Yaskawa INFORM job: ARGAZ.JBI

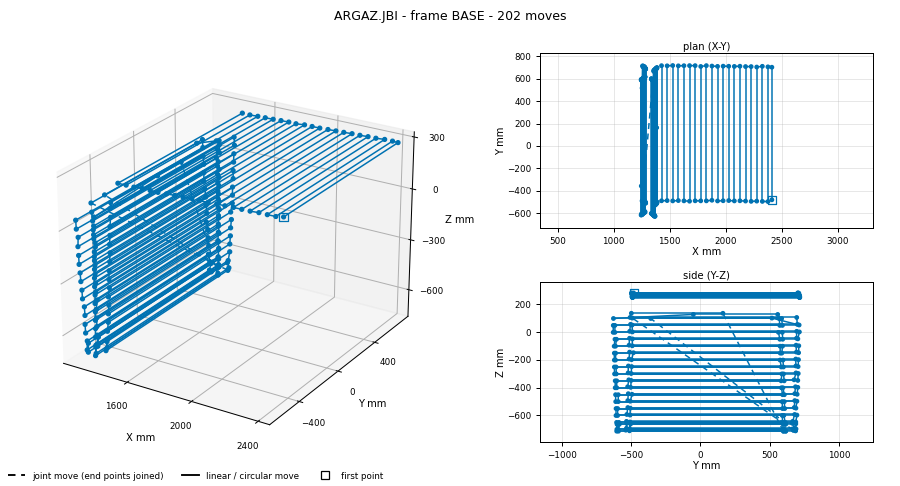
[picture p0: tool path of ARGAZ.JBI in frame BASE, 202 of 208 moves have a stored position in this frame; points joined in program order, loops and branches not executed]
/JOB
//NAME ARGAZ
//POS
///NPOS 202,0,202,0,0,0
///TOOL 0
///POSTYPE BASE
///RECTAN
///RCONF 1,0,0,0,0,0,0,0,0,0,0,0,0,0,0,0,0,0,0,0,0,0,0,0
C00000=2413.206274,-480.697971,282.313473,175.000000,5.000000,5.000000
C00001=2413.206274,703.166336,282.313473,175.000000,5.000000,5.000000
C00002=2378.104531,706.654151,282.437477,175.000000,5.000000,5.000000
C00003=2378.104531,-496.268820,282.437477,175.000000,5.000000,5.000000
C00004=2328.104531,-494.692713,280.280820,175.000000,5.000000,5.000000
C00005=2328.104531,711.367526,280.280820,175.000000,5.000000,5.000000
C00006=2278.104531,704.842987,278.975224,175.000000,5.000000,5.000000
C00007=2278.104531,-492.369314,278.975224,175.000000,5.000000,5.000000
C00008=2228.104531,-494.327219,276.432500,175.000000,5.000000,5.000000
C00009=2228.104531,708.877685,276.432500,175.000000,5.000000,5.000000
C00010=2178.104531,709.094399,273.988824,175.000000,5.000000,5.000000
C00011=2178.104531,-491.808166,273.988824,175.000000,5.000000,5.000000
C00012=2128.104531,-489.305417,272.087718,175.000000,5.000000,5.000000
C00013=2128.104531,712.128405,272.087718,175.000000,5.000000,5.000000
C00014=2078.104531,710.272403,270.104441,175.000000,5.000000,5.000000
C00015=2078.104531,-490.482062,270.104441,175.000000,5.000000,5.000000
C00016=2028.104531,-487.207564,267.676628,175.000000,5.000000,5.000000
C00017=2028.104531,711.894706,267.676628,175.000000,5.000000,5.000000
C00018=1978.104531,712.621618,265.646129,175.000000,5.000000,5.000000
C00019=1978.104531,-488.994271,265.646129,175.000000,5.000000,5.000000
C00020=1928.104531,-490.817664,264.262632,175.000000,5.000000,5.000000
C00021=1928.104531,710.764257,264.262632,175.000000,5.000000,5.000000
C00022=1878.104531,713.606685,262.597692,175.000000,5.000000,5.000000
C00023=1878.104531,-484.609026,262.597692,175.000000,5.000000,5.000000
C00024=1828.104531,-490.014665,260.699234,175.000000,5.000000,5.000000
C00025=1828.104531,717.443690,260.699234,175.000000,5.000000,5.000000
C00026=1778.104531,710.010172,259.433237,175.000000,5.000000,5.000000
C00027=1778.104531,-489.903250,259.433237,175.000000,5.000000,5.000000
C00028=1728.104531,-489.503789,257.000034,175.000000,5.000000,5.000000
C00029=1728.104531,717.230372,257.000034,175.000000,5.000000,5.000000
C00030=1678.104531,717.470864,255.326624,175.000000,5.000000,5.000000
C00031=1678.104531,-493.010626,255.326624,175.000000,5.000000,5.000000
C00032=1628.104531,-489.934501,253.475395,175.000000,5.000000,5.000000
C00033=1628.104531,716.829551,253.475395,175.000000,5.000000,5.000000
C00034=1578.104531,715.609427,252.672152,175.000000,5.000000,5.000000
C00035=1578.104531,-487.412050,252.672152,175.000000,5.000000,5.000000
C00036=1528.104531,-490.348908,250.461753,175.000000,5.000000,5.000000
C00037=1528.104531,718.341799,250.461753,175.000000,5.000000,5.000000
C00038=1478.104531,715.724918,249.387703,175.000000,5.000000,5.000000
C00039=1478.104531,-487.359740,249.387703,175.000000,5.000000,5.000000
C00040=1428.054088,-489.367917,249.591600,175.000000,5.000000,5.000000
C00041=1428.054088,717.087707,249.591600,175.000000,5.000000,5.000000
C00042=1375.381280,558.865130,127.297261,175.000000,-89.999999,5.000000
C00043=1375.381280,-49.872904,127.297261,175.000000,-89.999999,5.000000
C00044=1370.317972,-626.433977,98.135956,175.000000,-89.999999,5.000000
C00045=1370.317972,569.304121,98.135956,175.000000,-89.999999,5.000000
C00046=1368.165956,573.982169,48.135956,175.000000,-89.999999,5.000000
C00047=1368.165956,-627.765516,48.135956,175.000000,-89.999999,5.000000
C00048=1366.300613,-628.336175,-1.864044,175.000000,-89.999999,5.000000
C00049=1366.300613,564.146447,-1.864044,175.000000,-89.999999,5.000000
C00050=1364.709070,574.518860,-51.864044,175.000000,-89.999999,5.000000
C00051=1364.709070,-615.470524,-51.864044,175.000000,-89.999999,5.000000
C00052=1362.699081,-621.338804,-101.864044,175.000000,-89.999999,5.000000
C00053=1362.699081,576.164261,-101.864044,175.000000,-89.999999,5.000000
C00054=1361.029734,577.134382,-151.864044,175.000000,-89.999999,5.000000
C00055=1361.029734,-620.046668,-151.864044,175.000000,-89.999999,5.000000
C00056=1359.409458,-620.048027,-201.864044,175.000000,-89.999999,5.000000
C00057=1359.409458,575.847681,-201.864044,175.000000,-89.999999,5.000000
C00058=1357.613517,584.372245,-251.864044,175.000000,-89.999999,5.000000
C00059=1357.613517,-619.966504,-251.864044,175.000000,-89.999999,5.000000
C00060=1355.809114,-618.285777,-301.864044,175.000000,-89.999999,5.000000
C00061=1355.809114,588.836976,-301.864044,175.000000,-89.999999,5.000000
C00062=1353.972481,583.403483,-351.864044,175.000000,-89.999999,5.000000
C00063=1353.972481,-613.874036,-351.864044,175.000000,-89.999999,5.000000
C00064=1352.018958,-613.863166,-401.864044,175.000000,-89.999999,5.000000
C00065=1352.018958,585.494542,-401.864044,175.000000,-89.999999,5.000000
C00066=1350.088816,594.463405,-451.864044,175.000000,-89.999999,5.000000
C00067=1350.088816,-611.032968,-451.864044,175.000000,-89.999999,5.000000
C00068=1348.161110,-610.087304,-501.864044,175.000000,-89.999999,5.000000
C00069=1348.161110,590.588356,-501.864044,175.000000,-89.999999,5.000000
C00070=1346.094321,593.798995,-551.864044,175.000000,-89.999999,5.000000
C00071=1346.094321,-607.729937,-551.864044,175.000000,-89.999999,5.000000
C00072=1344.309797,-608.197334,-601.864044,175.000000,-89.999999,5.000000
C00073=1344.309797,591.908346,-601.864044,175.000000,-89.999999,5.000000
C00074=1342.380235,593.679428,-651.864044,175.000000,-89.999999,5.000000
C00075=1342.380235,-603.654478,-651.864044,175.000000,-89.999999,5.000000
C00076=1340.669129,-601.653773,-701.864044,175.000000,-89.999999,5.000000
C00077=1340.669129,595.156349,-701.864044,175.000000,-89.999999,5.000000
C00078=1338.968924,598.160463,-665.261503,180.000000,-60.000000,0.000000
C00079=1338.968924,-600.617076,-665.261503,180.000000,-60.000000,0.000000
C00080=1337.538666,-602.949985,-715.261503,180.000000,-60.000000,0.000000
C00081=1337.538666,600.315381,-715.261503,180.000000,-60.000000,0.000000
C00082=1337.538666,600.315381,-715.261503,180.000000,-60.000000,0.000000
C00083=1384.573264,163.476492,135.649179,175.000000,-89.999999,5.000000
C00084=1384.573264,-497.212784,135.649179,175.000000,-89.999999,5.000000
C00085=1387.134154,-506.685611,105.452428,175.000000,-89.999999,5.000000
C00086=1387.134154,696.005872,105.452428,175.000000,-89.999999,5.000000
C00087=1386.644943,700.400566,55.452428,175.000000,-89.999999,5.000000
C00088=1386.644943,-503.175845,55.452428,175.000000,-89.999999,5.000000
C00089=1385.416341,-509.347205,5.452428,175.000000,-89.999999,5.000000
C00090=1385.416341,695.993619,5.452428,175.000000,-89.999999,5.000000
C00091=1384.530286,694.673032,-44.547572,175.000000,-89.999999,5.000000
C00092=1384.530286,-510.215797,-44.547572,175.000000,-89.999999,5.000000
C00093=1383.211942,-513.702418,-94.547572,175.000000,-89.999999,5.000000
C00094=1383.211942,691.424661,-94.547572,175.000000,-89.999999,5.000000
C00095=1382.029329,693.773127,-144.547572,175.000000,-89.999999,5.000000
C00096=1382.029329,-510.105522,-144.547572,175.000000,-89.999999,5.000000
C00097=1380.742282,-513.419241,-194.547572,175.000000,-89.999999,5.000000
C00098=1380.742282,689.151074,-194.547572,175.000000,-89.999999,5.000000
C00099=1379.317619,689.923005,-244.547572,175.000000,-89.999999,5.000000
C00100=1379.317619,-518.588589,-244.547572,175.000000,-89.999999,5.000000
C00101=1377.622991,-520.482337,-294.547572,175.000000,-89.999999,5.000000
C00102=1377.622991,690.843331,-294.547572,175.000000,-89.999999,5.000000
C00103=1375.725701,676.986701,-344.547572,175.000000,-89.999999,5.000000
C00104=1375.725701,-515.830333,-344.547572,175.000000,-89.999999,5.000000
C00105=1373.930863,-523.962151,-394.547572,175.000000,-89.999999,5.000000
C00106=1373.930863,687.201507,-394.547572,175.000000,-89.999999,5.000000
C00107=1371.931878,682.022629,-444.547572,175.000000,-89.999999,5.000000
C00108=1371.931878,-519.291087,-444.547572,175.000000,-89.999999,5.000000
C00109=1370.288163,-523.069053,-494.547572,175.000000,-89.999999,5.000000
C00110=1370.288163,681.905546,-494.547572,175.000000,-89.999999,5.000000
C00111=1368.373992,678.466575,-544.547572,175.000000,-89.999999,5.000000
C00112=1368.373992,-522.809020,-544.547572,175.000000,-89.999999,5.000000
C00113=1366.288380,-529.990561,-594.547572,175.000000,-89.999999,5.000000
C00114=1366.288380,681.080520,-594.547572,175.000000,-89.999999,5.000000
C00115=1364.367259,667.085024,-644.547572,175.000000,-89.999999,5.000000
C00116=1364.367259,-532.326774,-644.547572,175.000000,-89.999999,5.000000
C00117=1362.423936,-532.694360,-694.547572,175.000000,-89.999999,5.000000
C00118=1362.423936,677.683753,-694.547572,175.000000,-89.999999,5.000000
C00119=1360.448293,664.032699,-657.945032,180.000000,-60.000000,0.000000
C00120=1360.448293,-528.686312,-657.945032,180.000000,-60.000000,0.000000
C00121=1358.736655,-537.636349,-707.945032,180.000000,-60.000000,0.000000
C00122=1358.736655,671.519200,-707.945032,180.000000,-60.000000,0.000000
C00123=1358.736655,671.519200,-707.945032,180.000000,-60.000000,0.000000
C00124=1254.346646,-489.805456,101.042867,175.000000,-89.999999,5.000000
C00125=1254.346646,517.104174,101.042867,175.000000,-89.999999,5.000000
C00126=1258.463174,713.476215,51.042867,175.000000,-89.999999,5.000000
C00127=1258.463174,-491.860509,51.042867,175.000000,-89.999999,5.000000
C00128=1261.233179,-489.734803,1.042867,175.000000,-89.999999,5.000000
C00129=1261.233179,715.246618,1.042867,175.000000,-89.999999,5.000000
C00130=1263.530822,704.150010,-48.957133,175.000000,-89.999999,5.000000
C00131=1263.530822,-489.611160,-48.957133,175.000000,-89.999999,5.000000
C00132=1265.803484,-490.551389,-98.957133,175.000000,-89.999999,5.000000
C00133=1265.803484,711.067217,-98.957133,175.000000,-89.999999,5.000000
C00134=1268.209382,709.711222,-148.957133,175.000000,-89.999999,5.000000
C00135=1268.209382,-482.270035,-148.957133,175.000000,-89.999999,5.000000
C00136=1269.839575,-495.608518,-198.957133,175.000000,-89.999999,5.000000
C00137=1269.839575,708.751971,-198.957133,175.000000,-89.999999,5.000000
C00138=1271.633535,706.020958,-248.957133,175.000000,-89.999999,5.000000
C00139=1271.633535,-495.046011,-248.957133,175.000000,-89.999999,5.000000
C00140=1273.209045,-498.528392,-298.957133,175.000000,-89.999999,5.000000
C00141=1273.209045,707.091624,-298.957133,175.000000,-89.999999,5.000000
C00142=1274.778950,703.821202,-348.957133,175.000000,-89.999999,5.000000
C00143=1274.778950,-498.652035,-348.957133,175.000000,-89.999999,5.000000
C00144=1276.502901,-501.906152,-398.957133,175.000000,-89.999999,5.000000
C00145=1276.502901,703.989682,-398.957133,175.000000,-89.999999,5.000000
C00146=1277.998844,699.262721,-448.957133,175.000000,-89.999999,5.000000
C00147=1277.998844,-492.101681,-448.957133,175.000000,-89.999999,5.000000
C00148=1279.424846,-505.182009,-498.957133,175.000000,-89.999999,5.000000
C00149=1279.424846,697.394490,-498.957133,175.000000,-89.999999,5.000000
C00150=1280.126954,690.352282,-548.957133,175.000000,-89.999999,5.000000
C00151=1280.126954,-504.584175,-548.957133,175.000000,-89.999999,5.000000
C00152=1281.384025,-506.767627,-598.957133,175.000000,-89.999999,5.000000
C00153=1281.384025,697.495035,-598.957133,175.000000,-89.999999,5.000000
C00154=1282.818366,689.325095,-648.957133,175.000000,-89.999999,5.000000
C00155=1282.818366,-506.682028,-648.957133,175.000000,-89.999999,5.000000
C00156=1284.126716,-509.875003,-698.957133,175.000000,-89.999999,5.000000
C00157=1284.126716,691.027562,-698.957133,175.000000,-89.999999,5.000000
C00158=1285.461074,689.375368,-662.354593,180.000000,-60.000000,0.000000
C00159=1285.461074,-501.749900,-662.354593,180.000000,-60.000000,0.000000
C00160=1286.533597,-510.586968,-712.354593,180.000000,-60.000000,0.000000
C00161=1286.533597,687.223167,-712.354593,180.000000,-60.000000,0.000000
C00162=1286.533597,687.223167,-712.354593,180.000000,-60.000000,0.000000
C00163=1247.184948,-357.258152,98.133703,175.000000,-89.999999,5.000000
C00164=1247.184948,587.097994,98.133703,175.000000,-89.999999,5.000000
C00165=1245.843306,592.746565,48.133703,175.000000,-89.999999,5.000000
C00166=1245.843306,-616.020977,48.133703,175.000000,-89.999999,5.000000
C00167=1247.718409,-615.852160,-1.866297,175.000000,-89.999999,5.000000
C00168=1247.718409,592.113501,-1.866297,175.000000,-89.999999,5.000000
C00169=1249.627062,594.663458,-51.866297,175.000000,-89.999999,5.000000
C00170=1249.627062,-604.746979,-51.866297,175.000000,-89.999999,5.000000
C00171=1251.401209,-611.430237,-101.866297,175.000000,-89.999999,5.000000
C00172=1251.401209,593.745855,-101.866297,175.000000,-89.999999,5.000000
C00173=1253.367892,588.365485,-151.866297,175.000000,-89.999999,5.000000
C00174=1253.367892,-610.535777,-151.866297,175.000000,-89.999999,5.000000
C00175=1255.139335,-611.488778,-201.866297,175.000000,-89.999999,5.000000
C00176=1255.139335,597.021454,-201.866297,175.000000,-89.999999,5.000000
C00177=1256.999427,599.889986,-251.866297,175.000000,-89.999999,5.000000
C00178=1256.999427,-607.499790,-251.866297,175.000000,-89.999999,5.000000
C00179=1259.062129,-606.254082,-301.866297,175.000000,-89.999999,5.000000
C00180=1259.062129,600.841625,-301.866297,175.000000,-89.999999,5.000000
C00181=1261.582176,605.514051,-351.866297,175.000000,-89.999999,5.000000
C00182=1261.582176,-602.829406,-351.866297,175.000000,-89.999999,5.000000
C00183=1263.639717,-602.839616,-401.866297,175.000000,-89.999999,5.000000
C00184=1263.639717,596.578989,-401.866297,175.000000,-89.999999,5.000000
C00185=1265.975009,606.745464,-451.866297,175.000000,-89.999999,5.000000
C00186=1265.975009,-591.829736,-451.866297,175.000000,-89.999999,5.000000
C00187=1268.177807,-591.867856,-501.866297,175.000000,-89.999999,5.000000
C00188=1268.177807,606.511299,-501.866297,175.000000,-89.999999,5.000000
C00189=1270.115574,609.444498,-551.866297,175.000000,-89.999999,5.000000
C00190=1270.115574,-596.282972,-551.866297,175.000000,-89.999999,5.000000
C00191=1272.145767,-596.372826,-601.866297,175.000000,-89.999999,5.000000
C00192=1272.145767,602.765325,-601.866297,175.000000,-89.999999,5.000000
C00193=1274.380461,613.267393,-651.866297,175.000000,-89.999999,5.000000
C00194=1274.380461,-586.885024,-651.866297,175.000000,-89.999999,5.000000
C00195=1276.674662,-593.241538,-701.866297,175.000000,-89.999999,5.000000
C00196=1276.674662,605.219983,-701.866297,175.000000,-89.999999,5.000000
C00197=1278.882309,616.568178,-665.263757,180.000000,-60.000000,0.000000
C00198=1278.882309,-584.132213,-665.263757,180.000000,-60.000000,0.000000
C00199=1281.187235,-589.960493,-715.263757,180.000000,-60.000000,0.000000
C00200=1281.187235,616.391873,-715.263757,180.000000,-60.000000,0.000000
C00201=1281.187235,616.391873,-715.263757,180.000000,-60.000000,0.000000
///POSTYPE PULSE
///PULSE
EC00000=0
EC00001=0
EC00002=0
EC00003=0
EC00004=0
EC00005=0
EC00006=0
EC00007=0
EC00008=0
EC00009=0
EC00010=0
EC00011=0
EC00012=0
EC00013=0
EC00014=0
EC00015=0
EC00016=0
EC00017=0
EC00018=0
EC00019=0
EC00020=0
EC00021=0
EC00022=0
EC00023=0
EC00024=0
EC00025=0
EC00026=0
EC00027=0
EC00028=0
EC00029=0
EC00030=0
EC00031=0
EC00032=0
EC00033=0
EC00034=0
EC00035=0
EC00036=0
EC00037=0
EC00038=0
EC00039=0
EC00040=0
EC00041=0
EC00042=0
EC00043=0
EC00044=0
EC00045=0
EC00046=0
EC00047=0
EC00048=0
EC00049=0
EC00050=0
EC00051=0
EC00052=0
EC00053=0
EC00054=0
EC00055=0
EC00056=0
EC00057=0
EC00058=0
EC00059=0
EC00060=0
EC00061=0
EC00062=0
EC00063=0
EC00064=0
EC00065=0
EC00066=0
EC00067=0
EC00068=0
EC00069=0
EC00070=0
EC00071=0
EC00072=0
EC00073=0
EC00074=0
EC00075=0
EC00076=0
EC00077=0
EC00078=0
EC00079=0
EC00080=0
EC00081=0
EC00082=92160
EC00083=92160
EC00084=92160
EC00085=92160
EC00086=92160
EC00087=92160
EC00088=92160
EC00089=92160
EC00090=92160
EC00091=92160
EC00092=92160
EC00093=92160
EC00094=92160
EC00095=92160
EC00096=92160
EC00097=92160
EC00098=92160
EC00099=92160
EC00100=92160
EC00101=92160
EC00102=92160
EC00103=92160
EC00104=92160
EC00105=92160
EC00106=92160
EC00107=92160
EC00108=92160
EC00109=92160
EC00110=92160
EC00111=92160
EC00112=92160
EC00113=92160
EC00114=92160
EC00115=92160
EC00116=92160
EC00117=92160
EC00118=92160
EC00119=92160
EC00120=92160
EC00121=92160
EC00122=92160
EC00123=184320
EC00124=184320
EC00125=184320
EC00126=184320
EC00127=184320
EC00128=184320
EC00129=184320
EC00130=184320
EC00131=184320
EC00132=184320
EC00133=184320
EC00134=184320
EC00135=184320
EC00136=184320
EC00137=184320
EC00138=184320
EC00139=184320
EC00140=184320
EC00141=184320
EC00142=184320
EC00143=184320
EC00144=184320
EC00145=184320
EC00146=184320
EC00147=184320
EC00148=184320
EC00149=184320
EC00150=184320
EC00151=184320
EC00152=184320
EC00153=184320
EC00154=184320
EC00155=184320
EC00156=184320
EC00157=184320
EC00158=184320
EC00159=184320
EC00160=184320
EC00161=184320
EC00162=276480
EC00163=276480
EC00164=276480
EC00165=276480
EC00166=276480
EC00167=276480
EC00168=276480
EC00169=276480
EC00170=276480
EC00171=276480
EC00172=276480
EC00173=276480
EC00174=276480
EC00175=276480
EC00176=276480
EC00177=276480
EC00178=276480
EC00179=276480
EC00180=276480
EC00181=276480
EC00182=276480
EC00183=276480
EC00184=276480
EC00185=276480
EC00186=276480
EC00187=276480
EC00188=276480
EC00189=276480
EC00190=276480
EC00191=276480
EC00192=276480
EC00193=276480
EC00194=276480
EC00195=276480
EC00196=276480
EC00197=276480
EC00198=276480
EC00199=276480
EC00200=276480
EC00201=368640
//INST
///DATE 2023/03/02 15:50
///ATTR SC,RW,RJ
////FRAME BASE
///GROUP1 RB1,ST1
NOP
MOVJ P009 EX000 VJ=15.00
MOVJ C00000 EC00000 VJ=15.0
CALL JOB:SPYON
MOVL C00001 EC00001 V=150.0
MOVL C00002 EC00002 V=150.0
MOVL C00003 EC00003 V=150.0
MOVL C00004 EC00004 V=150.0
MOVL C00005 EC00005 V=150.0
MOVL C00006 EC00006 V=150.0
MOVL C00007 EC00007 V=150.0
MOVL C00008 EC00008 V=150.0
MOVL C00009 EC00009 V=150.0
MOVL C00010 EC00010 V=150.0
MOVL C00011 EC00011 V=150.0
MOVL C00012 EC00012 V=150.0
MOVL C00013 EC00013 V=150.0
MOVL C00014 EC00014 V=150.0
MOVL C00015 EC00015 V=150.0
MOVL C00016 EC00016 V=150.0
MOVL C00017 EC00017 V=150.0
MOVL C00018 EC00018 V=150.0
MOVL C00019 EC00019 V=150.0
MOVL C00020 EC00020 V=150.0
MOVL C00021 EC00021 V=150.0
MOVL C00022 EC00022 V=150.0
MOVL C00023 EC00023 V=150.0
MOVL C00024 EC00024 V=150.0
MOVL C00025 EC00025 V=150.0
MOVL C00026 EC00026 V=150.0
MOVL C00027 EC00027 V=150.0
MOVL C00028 EC00028 V=150.0
MOVL C00029 EC00029 V=150.0
MOVL C00030 EC00030 V=150.0
MOVL C00031 EC00031 V=150.0
MOVL C00032 EC00032 V=150.0
MOVL C00033 EC00033 V=150.0
MOVL C00034 EC00034 V=150.0
MOVL C00035 EC00035 V=150.0
MOVL C00036 EC00036 V=150.0
MOVL C00037 EC00037 V=150.0
MOVL C00038 EC00038 V=150.0
MOVL C00039 EC00039 V=150.0
MOVL C00040 EC00040 V=150.0
MOVL C00041 EC00041 V=150.0
CALL JOB:SPYOF
MOVJ P009 VJ=15.00
MOVJ C00042 EC00042 VJ=15.0
CALL JOB:SPYON
MOVL C00043 EC00043 V=150.0
MOVL C00044 EC00044 V=150.0
MOVL C00045 EC00045 V=150.0
MOVL C00046 EC00046 V=150.0
MOVL C00047 EC00047 V=150.0
MOVL C00048 EC00048 V=150.0
MOVL C00049 EC00049 V=150.0
MOVL C00050 EC00050 V=150.0
MOVL C00051 EC00051 V=150.0
MOVL C00052 EC00052 V=150.0
MOVL C00053 EC00053 V=150.0
MOVL C00054 EC00054 V=150.0
MOVL C00055 EC00055 V=150.0
MOVL C00056 EC00056 V=150.0
MOVL C00057 EC00057 V=150.0
MOVL C00058 EC00058 V=150.0
MOVL C00059 EC00059 V=150.0
MOVL C00060 EC00060 V=150.0
MOVL C00061 EC00061 V=150.0
MOVL C00062 EC00062 V=150.0
MOVL C00063 EC00063 V=150.0
MOVL C00064 EC00064 V=150.0
MOVL C00065 EC00065 V=150.0
MOVL C00066 EC00066 V=150.0
MOVL C00067 EC00067 V=150.0
MOVL C00068 EC00068 V=150.0
MOVL C00069 EC00069 V=150.0
MOVL C00070 EC00070 V=150.0
MOVL C00071 EC00071 V=150.0
MOVL C00072 EC00072 V=150.0
MOVL C00073 EC00073 V=150.0
MOVL C00074 EC00074 V=150.0
MOVL C00075 EC00075 V=150.0
MOVL C00076 EC00076 V=150.0
MOVL C00077 EC00077 V=150.0
MOVL C00078 EC00078 V=150.0
MOVL C00079 EC00079 V=150.0
MOVL C00080 EC00080 V=150.0
MOVL C00081 EC00081 V=150.0
CALL JOB:SPYOF
MOVJ P009 VJ=15.00
MOVL C00082 EC00082 V=150.0
MOVJ C00083 EC00083 VJ=15.0
CALL JOB:SPYON
MOVL C00084 EC00084 V=150.0
MOVL C00085 EC00085 V=150.0
MOVL C00086 EC00086 V=150.0
MOVL C00087 EC00087 V=150.0
MOVL C00088 EC00088 V=150.0
MOVL C00089 EC00089 V=150.0
MOVL C00090 EC00090 V=150.0
MOVL C00091 EC00091 V=150.0
MOVL C00092 EC00092 V=150.0
MOVL C00093 EC00093 V=150.0
MOVL C00094 EC00094 V=150.0
MOVL C00095 EC00095 V=150.0
MOVL C00096 EC00096 V=150.0
MOVL C00097 EC00097 V=150.0
MOVL C00098 EC00098 V=150.0
MOVL C00099 EC00099 V=150.0
MOVL C00100 EC00100 V=150.0
MOVL C00101 EC00101 V=150.0
MOVL C00102 EC00102 V=150.0
MOVL C00103 EC00103 V=150.0
MOVL C00104 EC00104 V=150.0
MOVL C00105 EC00105 V=150.0
MOVL C00106 EC00106 V=150.0
MOVL C00107 EC00107 V=150.0
MOVL C00108 EC00108 V=150.0
MOVL C00109 EC00109 V=150.0
MOVL C00110 EC00110 V=150.0
MOVL C00111 EC00111 V=150.0
MOVL C00112 EC00112 V=150.0
MOVL C00113 EC00113 V=150.0
MOVL C00114 EC00114 V=150.0
MOVL C00115 EC00115 V=150.0
MOVL C00116 EC00116 V=150.0
MOVL C00117 EC00117 V=150.0
MOVL C00118 EC00118 V=150.0
MOVL C00119 EC00119 V=150.0
MOVL C00120 EC00120 V=150.0
MOVL C00121 EC00121 V=150.0
MOVL C00122 EC00122 V=150.0
CALL JOB:SPYOF
MOVJ P009 VJ=15.00
MOVL C00123 EC00123 V=150.0
MOVJ C00124 EC00124 VJ=15.0
CALL JOB:SPYON
MOVL C00125 EC00125 V=150.0
MOVL C00126 EC00126 V=150.0
MOVL C00127 EC00127 V=150.0
MOVL C00128 EC00128 V=150.0
MOVL C00129 EC00129 V=150.0
MOVL C00130 EC00130 V=150.0
MOVL C00131 EC00131 V=150.0
MOVL C00132 EC00132 V=150.0
MOVL C00133 EC00133 V=150.0
MOVL C00134 EC00134 V=150.0
MOVL C00135 EC00135 V=150.0
MOVL C00136 EC00136 V=150.0
MOVL C00137 EC00137 V=150.0
MOVL C00138 EC00138 V=150.0
MOVL C00139 EC00139 V=150.0
MOVL C00140 EC00140 V=150.0
MOVL C00141 EC00141 V=150.0
MOVL C00142 EC00142 V=150.0
MOVL C00143 EC00143 V=150.0
MOVL C00144 EC00144 V=150.0
MOVL C00145 EC00145 V=150.0
MOVL C00146 EC00146 V=150.0
MOVL C00147 EC00147 V=150.0
MOVL C00148 EC00148 V=150.0
MOVL C00149 EC00149 V=150.0
MOVL C00150 EC00150 V=150.0
MOVL C00151 EC00151 V=150.0
MOVL C00152 EC00152 V=150.0
MOVL C00153 EC00153 V=150.0
MOVL C00154 EC00154 V=150.0
MOVL C00155 EC00155 V=150.0
MOVL C00156 EC00156 V=150.0
MOVL C00157 EC00157 V=150.0
MOVL C00158 EC00158 V=150.0
MOVL C00159 EC00159 V=150.0
MOVL C00160 EC00160 V=150.0
MOVL C00161 EC00161 V=150.0
CALL JOB:SPYOF
MOVJ P009 VJ=15.00
MOVL C00162 EC00162 V=150.0
MOVJ C00163 EC00163 VJ=15.0
CALL JOB:SPYON
MOVL C00164 EC00164 V=150.0
MOVL C00165 EC00165 V=150.0
MOVL C00166 EC00166 V=150.0
MOVL C00167 EC00167 V=150.0
MOVL C00168 EC00168 V=150.0
MOVL C00169 EC00169 V=150.0
MOVL C00170 EC00170 V=150.0
MOVL C00171 EC00171 V=150.0
MOVL C00172 EC00172 V=150.0
MOVL C00173 EC00173 V=150.0
MOVL C00174 EC00174 V=150.0
MOVL C00175 EC00175 V=150.0
MOVL C00176 EC00176 V=150.0
MOVL C00177 EC00177 V=150.0
MOVL C00178 EC00178 V=150.0
MOVL C00179 EC00179 V=150.0
MOVL C00180 EC00180 V=150.0
MOVL C00181 EC00181 V=150.0
MOVL C00182 EC00182 V=150.0
MOVL C00183 EC00183 V=150.0
MOVL C00184 EC00184 V=150.0
MOVL C00185 EC00185 V=150.0
MOVL C00186 EC00186 V=150.0
MOVL C00187 EC00187 V=150.0
MOVL C00188 EC00188 V=150.0
MOVL C00189 EC00189 V=150.0
MOVL C00190 EC00190 V=150.0
MOVL C00191 EC00191 V=150.0
MOVL C00192 EC00192 V=150.0
MOVL C00193 EC00193 V=150.0
MOVL C00194 EC00194 V=150.0
MOVL C00195 EC00195 V=150.0
MOVL C00196 EC00196 V=150.0
MOVL C00197 EC00197 V=150.0
MOVL C00198 EC00198 V=150.0
MOVL C00199 EC00199 V=150.0
MOVL C00200 EC00200 V=150.0
CALL JOB:SPYOF
MOVJ P009 VJ=15.00
MOVL C00201 EC00201 V=150.0
END
